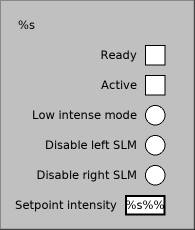
VISUALIZATION _VISU_UvLedModule  // 195x230
VAR_IN_OUT
  m_Inst_Fb   : FB_UvLedModule;
END_VAR
    Rectangle (0,0 195x230), colour variable: m_Inst_Fb._nColorRGB
        p2167032090: m_Inst_Fb._nColorRGB
        p3092690914: 16#FFFF0000
        p3450524324: 16#FF000000
    Rectangle (15,15 155x20), "%s", text variable: m_Inst_Fb._sColorName
    RoundedRectangle (145,45 20x20), colour toggle: m_Inst_Fb.IbReady
    Rectangle (20,45 120x20), "Ready"
    RoundedRectangle (145,75 20x20), colour toggle: m_Inst_Fb._bActivate
    Rectangle (20,75 120x20), "Active"
    Ellipse (145,105 20x20), colour toggle: m_Inst_Fb.RbLowIntenseMode
        toggle m_Inst_Fb.RbLowIntenseMode
    Rectangle (20,105 120x20), "Low intense mode"
    Ellipse (145,135 20x20), colour toggle: m_Inst_Fb.RbDisableLeft
        toggle m_Inst_Fb.RbDisableLeft
    Rectangle (20,135 120x20), "Disable left SLM"
    Ellipse (145,165 20x20), colour toggle: m_Inst_Fb.RbDisableRight
        toggle m_Inst_Fb.RbDisableRight
    Rectangle (20,165 120x20), "Disable right SLM"
    Rectangle (11,195 109x20), "Setpoint intensity"
    Rectangle (125,195 40x20), "%s%%", text variable: m_Inst_Fb.RnIntensitySetpoint
        OnMouseDown: write the text variable via VisuDialogs.Numpad, min m_Inst_Fb.CnMinIntensitySetpoint, max m_Inst_Fb.CnMaxIntensitySetpoint
END_VISUALIZATION

(* stored: Version 1.1.0.1, ProductVersion 3.1.4024.11
   Visu _VISU_UvLedModule: Id {491a0126-22dd-42e7-a326-7169338bbe07} *)
